INTERFACE PUBLIC ClearedStateCommands EXTENDS __System.IQueryInterface

METHOD PUBLIC Abort
END_METHOD

END_INTERFACE

(* stored: Version 1.1.0.1, ProductVersion 3.1.4026.18
   Itf ClearedStateCommands: Id {e37a0826-6562-0f43-3b89-25b56eaa6db9}
   Method Abort: Id {0a18bd59-645a-0630-0a33-290af6af5463} *)
